      A     M      0.2;
      =     L     22.0;
      BLD   103;
      AN    M      3.3;
      =     L     22.1;
      BLD   103;
      CALL FB    12 , DB    72 (
           REQ                      := L     22.0,
           R                        := L     22.1,
           ID                       := W#16#12,
           R_ID                     := DW#16#12,
           DONE                     := DB2.DBX   10.0,
           ERROR                    := DB2.DBX   10.1,
           STATUS                   := DB2.DBW   12,
           SD_1                     := DB16.SHUTTLE,
           LEN                      := #SEND2_LEN);
      NOP   0;
NETWORK
TITLE =

      L     20;
      T     #RECV3_LEN;
      NOP   0;
NETWORK
TITLE =LOCAL(CPU4) --> LOCAL(CPU3) 공정상태
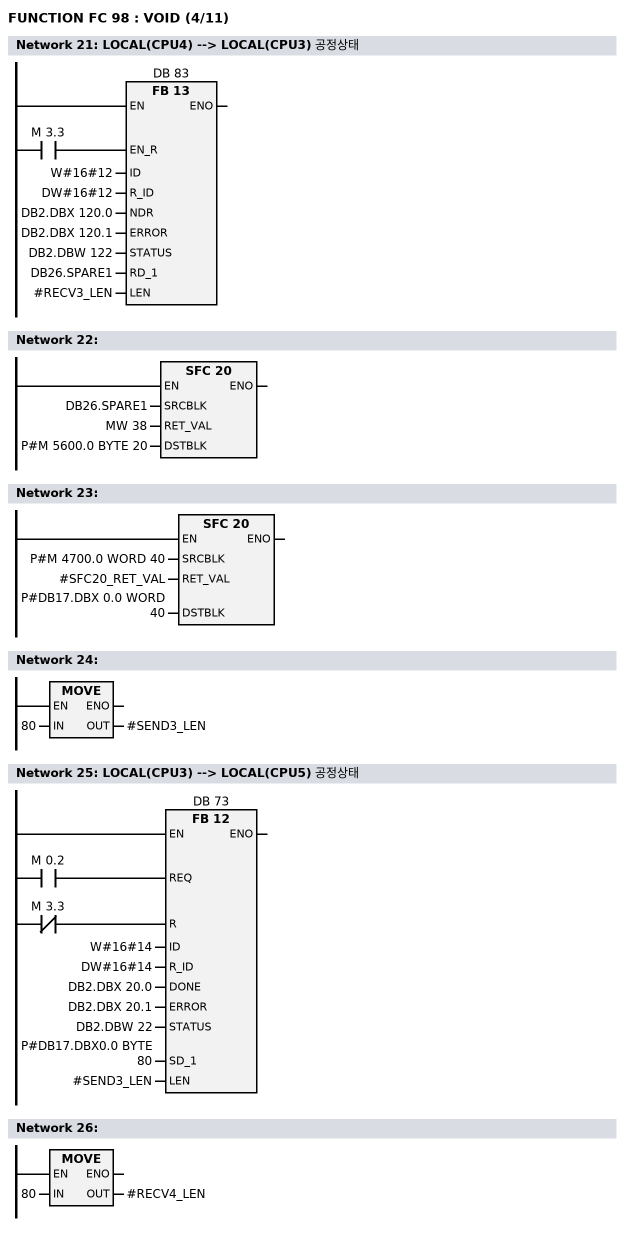

      A     M      3.3;
      =     L     22.0;
      BLD   103;
      CALL FB    13 , DB    83 (
           EN_R                     := L     22.0,
           ID                       := W#16#12,
           R_ID                     := DW#16#12,
           NDR                      := DB2.DBX  120.0,
           ERROR                    := DB2.DBX  120.1,
           STATUS                   := DB2.DBW  122,
           RD_1                     := DB26.SPARE1,
           LEN                      := #RECV3_LEN);
      NOP   0;
NETWORK
TITLE =

      CALL SFC   20 (
           SRCBLK                   := DB26.SPARE1,
           RET_VAL                  := MW    38,
           DSTBLK                   := P#M 5600.0 BYTE 20);
      NOP   0;
NETWORK
TITLE =

      CALL SFC   20 (
           SRCBLK                   := P#M 4700.0 WORD 40,
           RET_VAL                  := #SFC20_RET_VAL,
           DSTBLK                   := P#DB17.DBX 0.0 WORD 40);
      NOP   0;
NETWORK
TITLE =

      L     80;
      T     #SEND3_LEN;
      NOP   0;
NETWORK
TITLE =LOCAL(CPU3) --> LOCAL(CPU5) 공정상태

      A     M      0.2;
      =     L     22.0;
      BLD   103;
      AN    M      3.3;
      =     L     22.1;
      BLD   103;
      CALL FB    12 , DB    73 (
           REQ                      := L     22.0,
           R                        := L     22.1,
           ID                       := W#16#14,
           R_ID                     := DW#16#14,
           DONE                     := DB2.DBX   20.0,
           ERROR                    := DB2.DBX   20.1,
           STATUS                   := DB2.DBW   22,
           SD_1                     := P#DB17.DBX0.0 BYTE 80,
           LEN                      := #SEND3_LEN);
      NOP   0;
NETWORK
TITLE =

      L     80;
      T     #RECV4_LEN;
      NOP   0;
NETWORK
TITLE =LOCAL(CPU5) --> LOCAL(CPU3) 공정상태
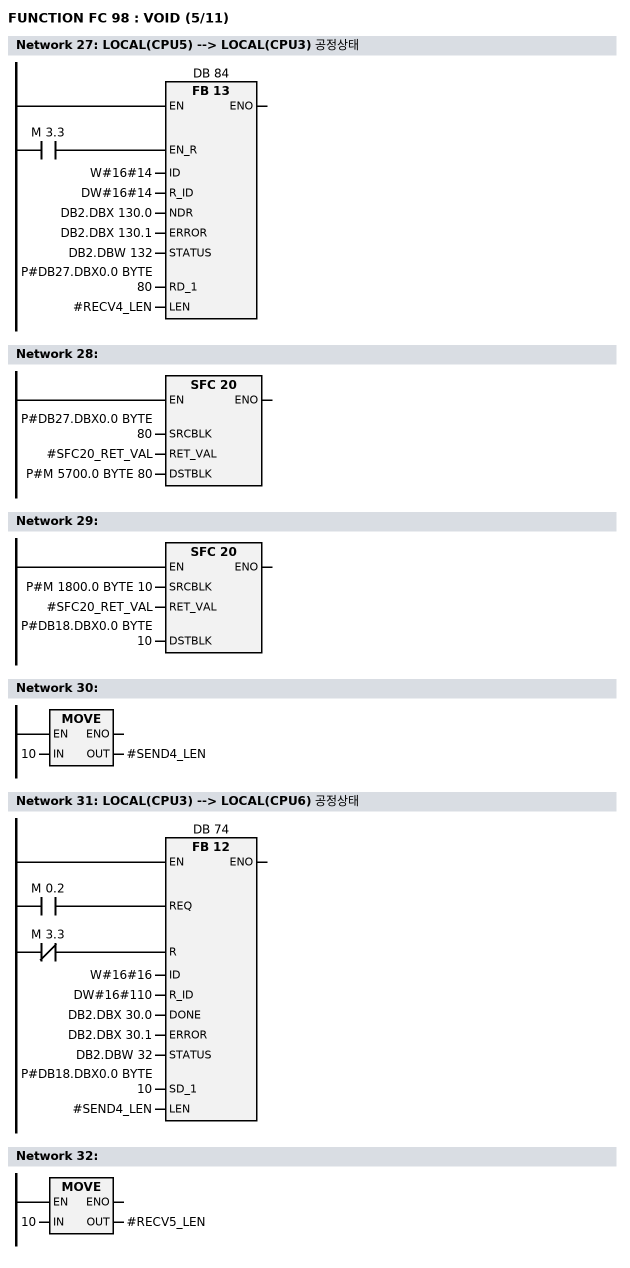

      A     M      3.3;
      =     L     22.0;
      BLD   103;
      CALL FB    13 , DB    84 (
           EN_R                     := L     22.0,
           ID                       := W#16#14,
           R_ID                     := DW#16#14,
           NDR                      := DB2.DBX  130.0,
           ERROR                    := DB2.DBX  130.1,
           STATUS                   := DB2.DBW  132,
           RD_1                     := P#DB27.DBX0.0 BYTE 80,
           LEN                      := #RECV4_LEN);
      NOP   0;
NETWORK
TITLE =

      CALL SFC   20 (
           SRCBLK                   := P#DB27.DBX0.0 BYTE 80,
           RET_VAL                  := #SFC20_RET_VAL,
           DSTBLK                   := P#M 5700.0 BYTE 80);
      NOP   0;
NETWORK
TITLE =

      CALL SFC   20 (
           SRCBLK                   := P#M 1800.0 BYTE 10,
           RET_VAL                  := #SFC20_RET_VAL,
           DSTBLK                   := P#DB18.DBX0.0 BYTE 10);
      NOP   0;
NETWORK
TITLE =

      L     10;
      T     #SEND4_LEN;
      NOP   0;
NETWORK
TITLE =LOCAL(CPU3) --> LOCAL(CPU6) 공정상태

      A     M      0.2;
      =     L     22.0;
      BLD   103;
      AN    M      3.3;
      =     L     22.1;
      BLD   103;
      CALL FB    12 , DB    74 (
           REQ                      := L     22.0,
           R                        := L     22.1,
           ID                       := W#16#16,
           R_ID                     := DW#16#110,
           DONE                     := DB2.DBX   30.0,
           ERROR                    := DB2.DBX   30.1,
           STATUS                   := DB2.DBW   32,
           SD_1                     := P#DB18.DBX0.0 BYTE 10,
           LEN                      := #SEND4_LEN);
      NOP   0;
NETWORK
TITLE =

      L     10;
      T     #RECV5_LEN;
      NOP   0;
NETWORK
TITLE =LOCAL(CPU6) --> LOCAL(CPU3) 공정상태
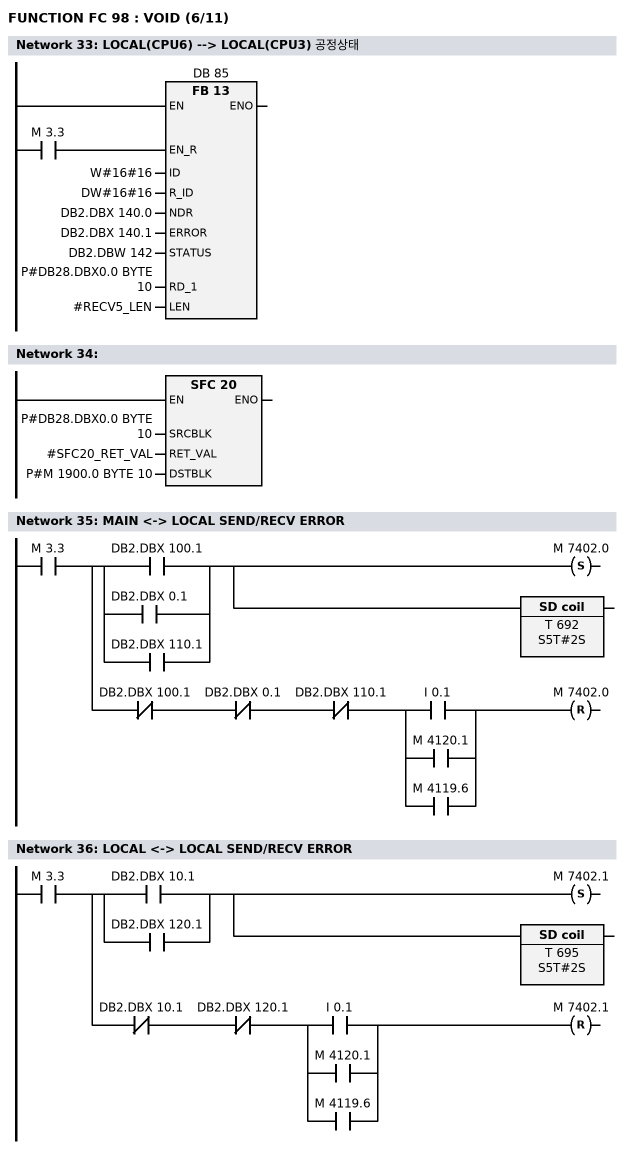

      A     M      3.3;
      =     L     22.0;
      BLD   103;
      CALL FB    13 , DB    85 (
           EN_R                     := L     22.0,
           ID                       := W#16#16,
           R_ID                     := DW#16#16,
           NDR                      := DB2.DBX  140.0,
           ERROR                    := DB2.DBX  140.1,
           STATUS                   := DB2.DBW  142,
           RD_1                     := P#DB28.DBX0.0 BYTE 10,
           LEN                      := #RECV5_LEN);
      NOP   0;
NETWORK
TITLE =

      CALL SFC   20 (
           SRCBLK                   := P#DB28.DBX0.0 BYTE 10,
           RET_VAL                  := #SFC20_RET_VAL,
           DSTBLK                   := P#M 1900.0 BYTE 10);
      NOP   0;
NETWORK
TITLE =MAIN <-> LOCAL SEND/RECV ERROR

      A     M      3.3;
      =     L     22.0;
      A     L     22.0;
      A(    ;
      O     DB2.DBX  100.1;
      O     DB2.DBX    0.1;
      O     DB2.DBX  110.1;
      )     ;
      S     M   7402.0;
      L     S5T#2S;
      SD    T    692;
      A     L     22.0;
      AN    DB2.DBX  100.1;
      AN    DB2.DBX    0.1;
      AN    DB2.DBX  110.1;
      A(    ;
      O     I      0.1;
      O     M   4120.1;
      O     M   4119.6;
      )     ;
      R     M   7402.0;
NETWORK
TITLE =LOCAL <-> LOCAL SEND/RECV ERROR

      A     M      3.3;
      =     L     22.0;
      A     L     22.0;
      A(    ;
      O     DB2.DBX   10.1;
      O     DB2.DBX  120.1;
      )     ;
      S     M   7402.1;
      L     S5T#2S;
      SD    T    695;
      A     L     22.0;
      AN    DB2.DBX   10.1;
      AN    DB2.DBX  120.1;
      A(    ;
      O     I      0.1;
      O     M   4120.1;
      O     M   4119.6;
      )     ;
      R     M   7402.1;
NETWORK
TITLE =LOCAL <-> LOCAL SEND/RECV ERROR
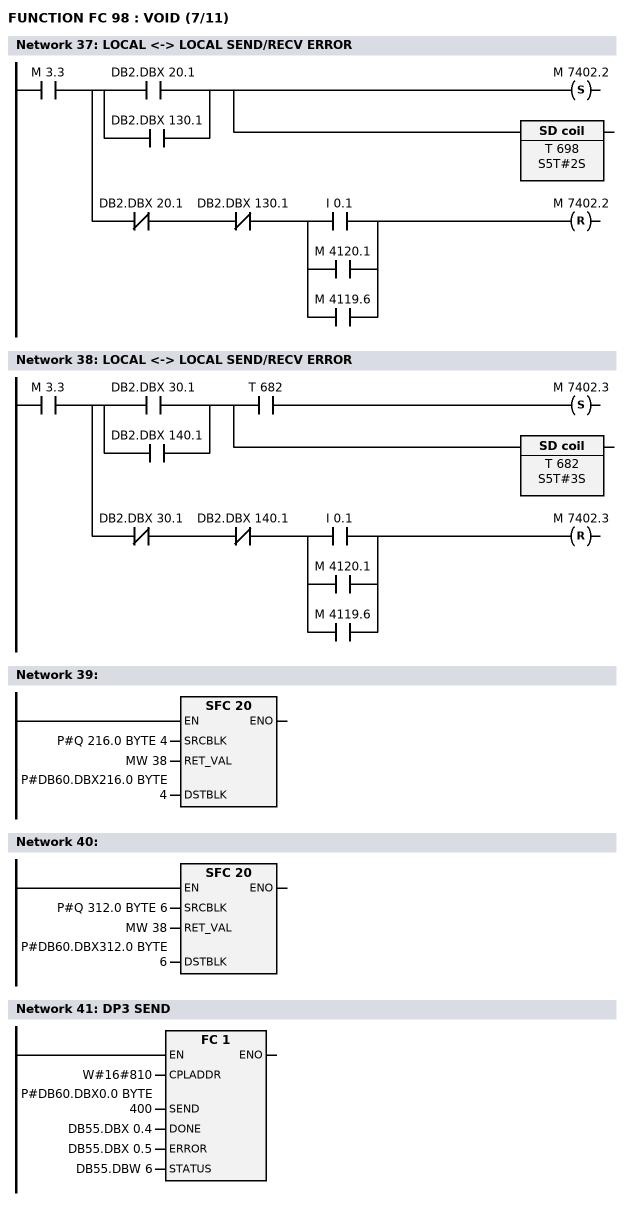

      A     M      3.3;
      =     L     22.0;
      A     L     22.0;
      A(    ;
      O     DB2.DBX   20.1;
      O     DB2.DBX  130.1;
      )     ;
      S     M   7402.2;
      L     S5T#2S;
      SD    T    698;
      A     L     22.0;
      AN    DB2.DBX   20.1;
      AN    DB2.DBX  130.1;
      A(    ;
      O     I      0.1;
      O     M   4120.1;
      O     M   4119.6;
      )     ;
      R     M   7402.2;
NETWORK
TITLE =LOCAL <-> LOCAL SEND/RECV ERROR

      A     M      3.3;
      =     L     22.0;
      A     L     22.0;
      A(    ;
      O     DB2.DBX   30.1;
      O     DB2.DBX  140.1;
      )     ;
      =     L     22.1;
      A     L     22.1;
      A     T    682;
      S     M   7402.3;
      A     L     22.1;
      BLD   102;
      L     S5T#3S;
      SD    T    682;
      A     L     22.0;
      AN    DB2.DBX   30.1;
      AN    DB2.DBX  140.1;
      A(    ;
      O     I      0.1;
      O     M   4120.1;
      O     M   4119.6;
      )     ;
      R     M   7402.3;
NETWORK
TITLE =

      CALL SFC   20 (
           SRCBLK                   := P#Q 216.0 BYTE 4,
           RET_VAL                  := MW    38,
           DSTBLK                   := P#DB60.DBX216.0 BYTE 4);
      NOP   0;
NETWORK
TITLE =

      CALL SFC   20 (
           SRCBLK                   := P#Q 312.0 BYTE 6,
           RET_VAL                  := MW    38,
           DSTBLK                   := P#DB60.DBX312.0 BYTE 6);
      NOP   0;
NETWORK
TITLE =DP3 SEND

      CALL FC     1 (
           CPLADDR                  := W#16#810,
           SEND                     := P#DB60.DBX0.0 BYTE 400,
           DONE                     := DB55.DBX    0.4,
           ERROR                    := DB55.DBX    0.5,
           STATUS                   := DB55.DBW    6);
      NOP   0;
NETWORK
TITLE =DP3 RECV
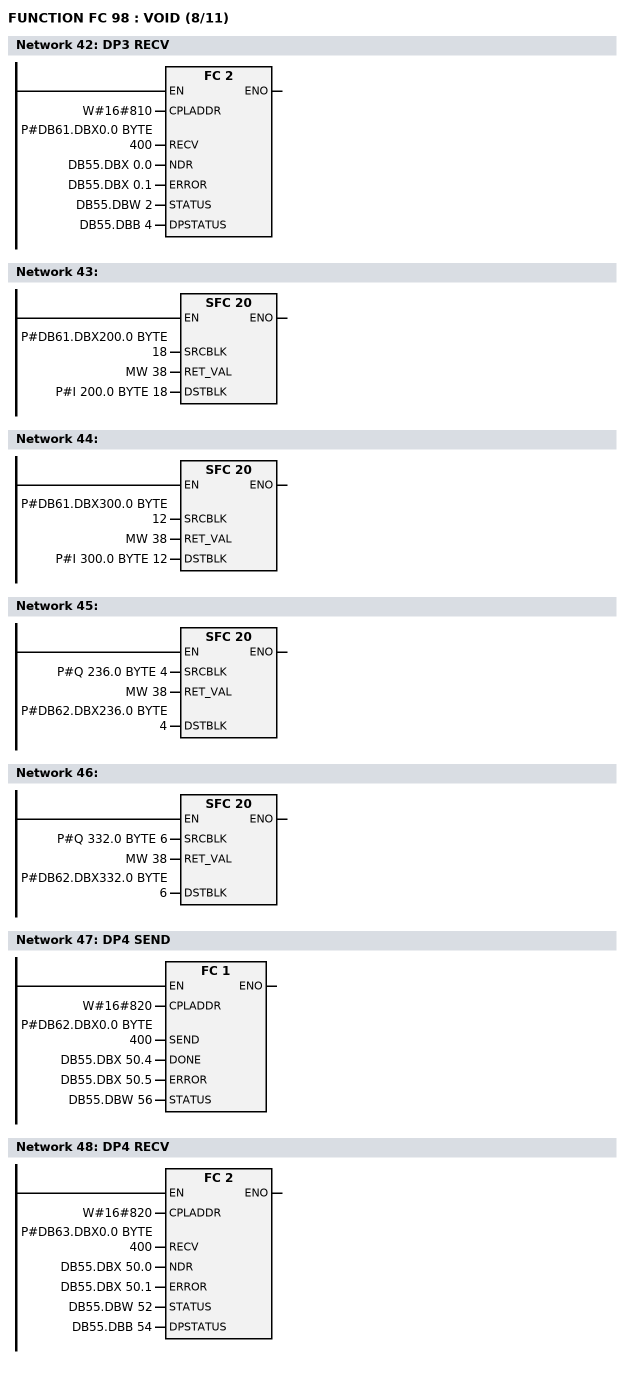

      CALL FC     2 (
           CPLADDR                  := W#16#810,
           RECV                     := P#DB61.DBX0.0 BYTE 400,
           NDR                      := DB55.DBX    0.0,
           ERROR                    := DB55.DBX    0.1,
           STATUS                   := DB55.DBW    2,
           DPSTATUS                 := DB55.DBB    4);
      NOP   0;
NETWORK
TITLE =

      CALL SFC   20 (
           SRCBLK                   := P#DB61.DBX200.0 BYTE 18,
           RET_VAL                  := MW    38,
           DSTBLK                   := P#I 200.0 BYTE 18);
      NOP   0;
NETWORK
TITLE =

      CALL SFC   20 (
           SRCBLK                   := P#DB61.DBX300.0 BYTE 12,
           RET_VAL                  := MW    38,
           DSTBLK                   := P#I 300.0 BYTE 12);
      NOP   0;
NETWORK
TITLE =

      CALL SFC   20 (
           SRCBLK                   := P#Q 236.0 BYTE 4,
           RET_VAL                  := MW    38,
           DSTBLK                   := P#DB62.DBX236.0 BYTE 4);
      NOP   0;
NETWORK
TITLE =

      CALL SFC   20 (
           SRCBLK                   := P#Q 332.0 BYTE 6,
           RET_VAL                  := MW    38,
           DSTBLK                   := P#DB62.DBX332.0 BYTE 6);
      NOP   0;
NETWORK
TITLE =DP4 SEND

      CALL FC     1 (
           CPLADDR                  := W#16#820,
           SEND                     := P#DB62.DBX0.0 BYTE 400,
           DONE                     := DB55.DBX   50.4,
           ERROR                    := DB55.DBX   50.5,
           STATUS                   := DB55.DBW   56);
      NOP   0;
NETWORK
TITLE =DP4 RECV

      CALL FC     2 (
           CPLADDR                  := W#16#820,
           RECV                     := P#DB63.DBX0.0 BYTE 400,
           NDR                      := DB55.DBX   50.0,
           ERROR                    := DB55.DBX   50.1,
           STATUS                   := DB55.DBW   52,
           DPSTATUS                 := DB55.DBB   54);
      NOP   0;
NETWORK
TITLE =
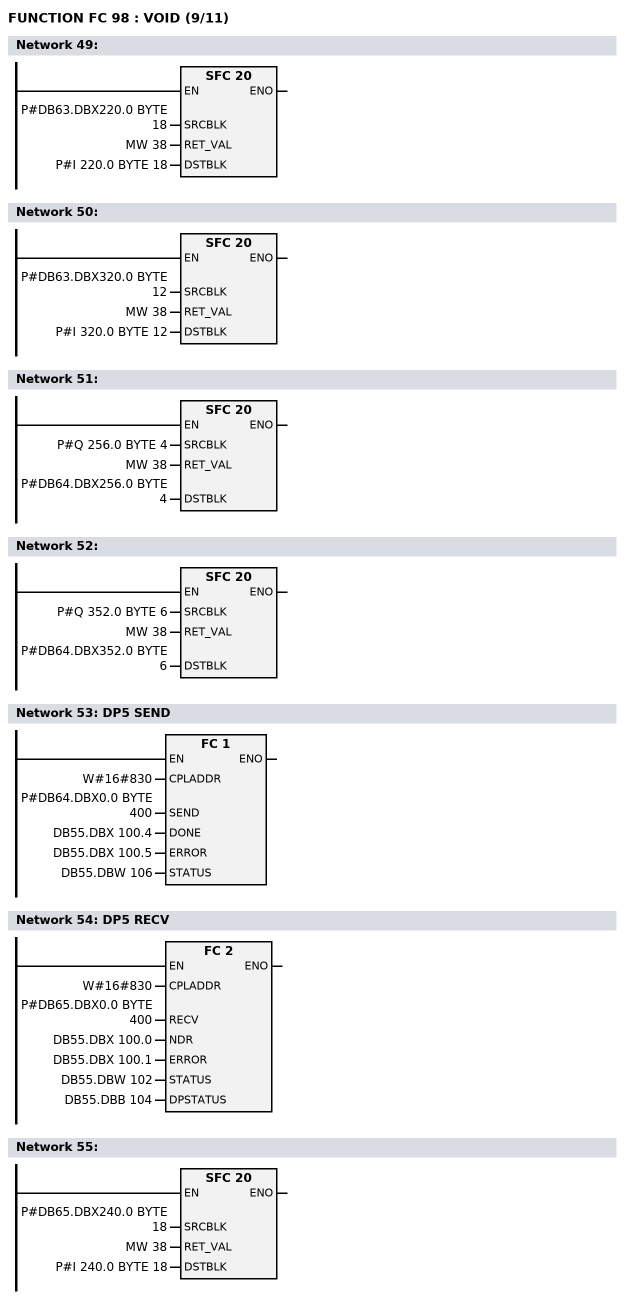

      CALL SFC   20 (
           SRCBLK                   := P#DB63.DBX220.0 BYTE 18,
           RET_VAL                  := MW    38,
           DSTBLK                   := P#I 220.0 BYTE 18);
      NOP   0;
NETWORK
TITLE =

      CALL SFC   20 (
           SRCBLK                   := P#DB63.DBX320.0 BYTE 12,
           RET_VAL                  := MW    38,
           DSTBLK                   := P#I 320.0 BYTE 12);
      NOP   0;
NETWORK
TITLE =

      CALL SFC   20 (
           SRCBLK                   := P#Q 256.0 BYTE 4,
           RET_VAL                  := MW    38,
           DSTBLK                   := P#DB64.DBX256.0 BYTE 4);
      NOP   0;
NETWORK
TITLE =

      CALL SFC   20 (
           SRCBLK                   := P#Q 352.0 BYTE 6,
           RET_VAL                  := MW    38,
           DSTBLK                   := P#DB64.DBX352.0 BYTE 6);
      NOP   0;
NETWORK
TITLE =DP5 SEND

      CALL FC     1 (
           CPLADDR                  := W#16#830,
           SEND                     := P#DB64.DBX0.0 BYTE 400,
           DONE                     := DB55.DBX  100.4,
           ERROR                    := DB55.DBX  100.5,
           STATUS                   := DB55.DBW  106);
      NOP   0;
NETWORK
TITLE =DP5 RECV

      CALL FC     2 (
           CPLADDR                  := W#16#830,
           RECV                     := P#DB65.DBX0.0 BYTE 400,
           NDR                      := DB55.DBX  100.0,
           ERROR                    := DB55.DBX  100.1,
           STATUS                   := DB55.DBW  102,
           DPSTATUS                 := DB55.DBB  104);
      NOP   0;
NETWORK
TITLE =

      CALL SFC   20 (
           SRCBLK                   := P#DB65.DBX240.0 BYTE 18,
           RET_VAL                  := MW    38,
           DSTBLK                   := P#I 240.0 BYTE 18);
      NOP   0;
NETWORK
TITLE =
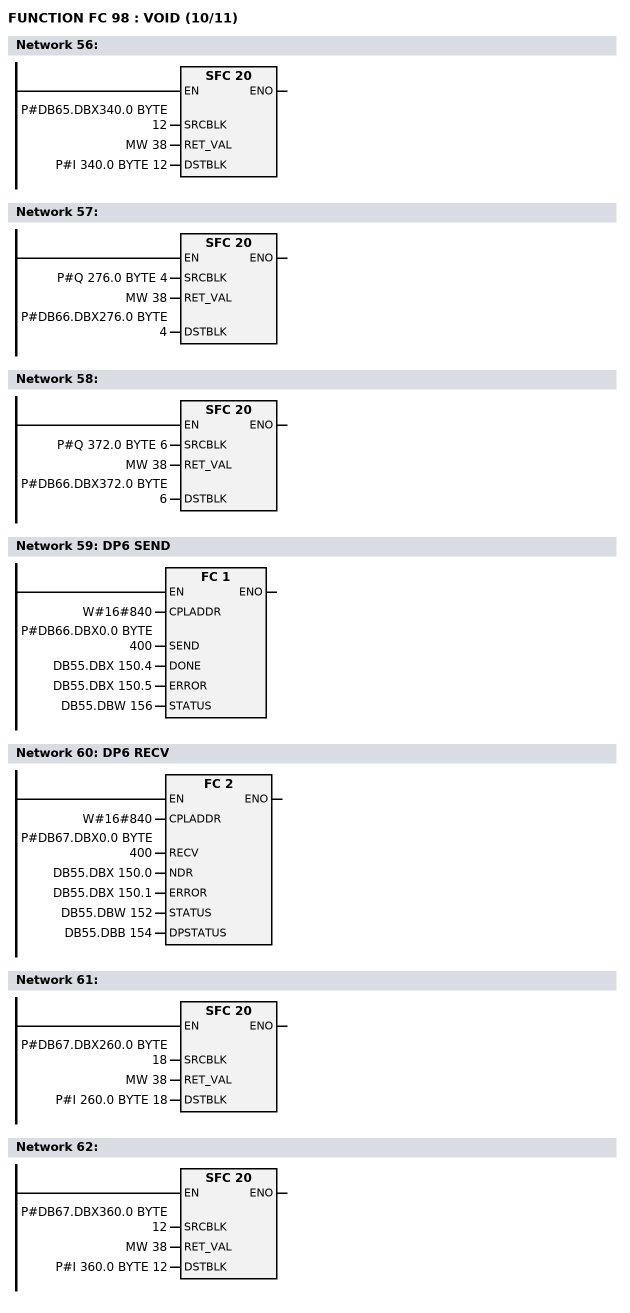

      CALL SFC   20 (
           SRCBLK                   := P#DB65.DBX340.0 BYTE 12,
           RET_VAL                  := MW    38,
           DSTBLK                   := P#I 340.0 BYTE 12);
      NOP   0;
NETWORK
TITLE =

      CALL SFC   20 (
           SRCBLK                   := P#Q 276.0 BYTE 4,
           RET_VAL                  := MW    38,
           DSTBLK                   := P#DB66.DBX276.0 BYTE 4);
      NOP   0;
NETWORK
TITLE =

      CALL SFC   20 (
           SRCBLK                   := P#Q 372.0 BYTE 6,
           RET_VAL                  := MW    38,
           DSTBLK                   := P#DB66.DBX372.0 BYTE 6);
      NOP   0;
NETWORK
TITLE =DP6 SEND

      CALL FC     1 (
           CPLADDR                  := W#16#840,
           SEND                     := P#DB66.DBX0.0 BYTE 400,
           DONE                     := DB55.DBX  150.4,
           ERROR                    := DB55.DBX  150.5,
           STATUS                   := DB55.DBW  156);
      NOP   0;
NETWORK
TITLE =DP6 RECV

      CALL FC     2 (
           CPLADDR                  := W#16#840,
           RECV                     := P#DB67.DBX0.0 BYTE 400,
           NDR                      := DB55.DBX  150.0,
           ERROR                    := DB55.DBX  150.1,
           STATUS                   := DB55.DBW  152,
           DPSTATUS                 := DB55.DBB  154);
      NOP   0;
NETWORK
TITLE =

      CALL SFC   20 (
           SRCBLK                   := P#DB67.DBX260.0 BYTE 18,
           RET_VAL                  := MW    38,
           DSTBLK                   := P#I 260.0 BYTE 18);
      NOP   0;
NETWORK
TITLE =

      CALL SFC   20 (
           SRCBLK                   := P#DB67.DBX360.0 BYTE 12,
           RET_VAL                  := MW    38,
           DSTBLK                   := P#I 360.0 BYTE 12);
      NOP   0;
NETWORK
TITLE =
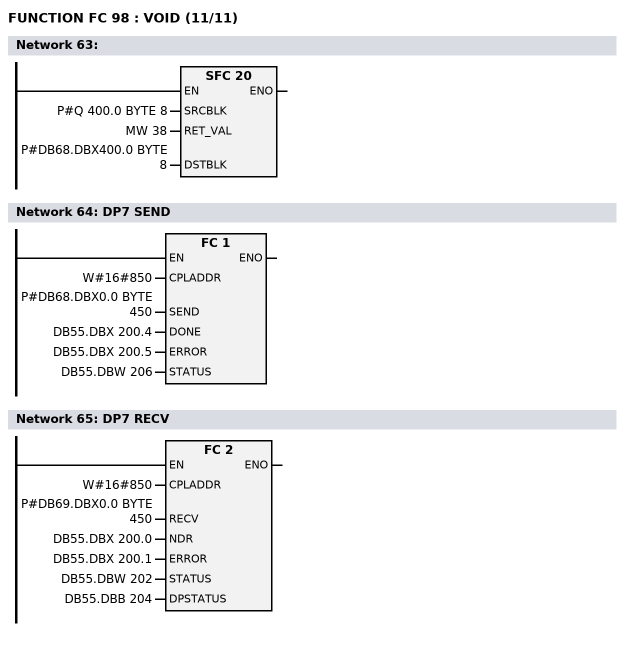

      CALL SFC   20 (
           SRCBLK                   := P#Q 400.0 BYTE 8,
           RET_VAL                  := MW    38,
           DSTBLK                   := P#DB68.DBX400.0 BYTE 8);
      NOP   0;
NETWORK
TITLE =DP7 SEND

      CALL FC     1 (
           CPLADDR                  := W#16#850,
           SEND                     := P#DB68.DBX0.0 BYTE 450,
           DONE                     := DB55.DBX  200.4,
           ERROR                    := DB55.DBX  200.5,
           STATUS                   := DB55.DBW  206);
      NOP   0;
NETWORK
TITLE =DP7 RECV

      CALL FC     2 (
           CPLADDR                  := W#16#850,
           RECV                     := P#DB69.DBX0.0 BYTE 450,
           NDR                      := DB55.DBX  200.0,
           ERROR                    := DB55.DBX  200.1,
           STATUS                   := DB55.DBW  202,
           DPSTATUS                 := DB55.DBB  204);
      NOP   0;
END_FUNCTION

FUNCTION FC 100 : VOID
TITLE =
VERSION : 0.1

BEGIN
NETWORK
TITLE =
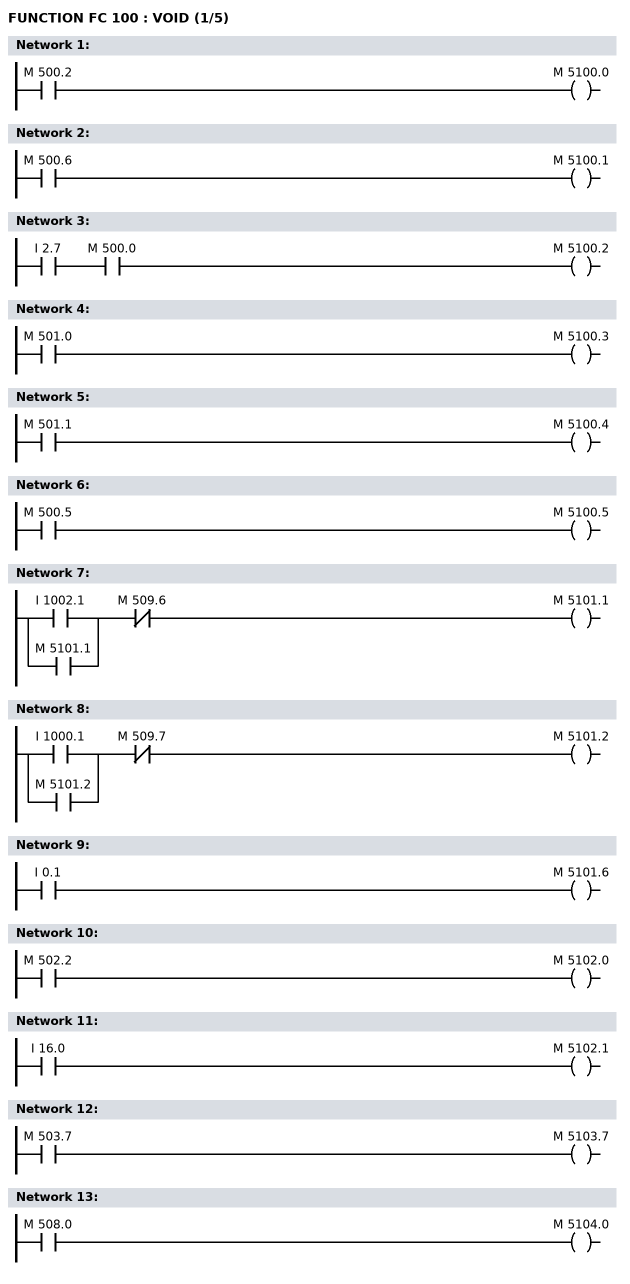

      A     M    500.2;
      =     M   5100.0;
NETWORK
TITLE =

      A     M    500.6;
      =     M   5100.1;
NETWORK
TITLE =

      A     I      2.7;
      A     M    500.0;
      =     M   5100.2;
NETWORK
TITLE =

      A     M    501.0;
      =     M   5100.3;
NETWORK
TITLE =

      A     M    501.1;
      =     M   5100.4;
NETWORK
TITLE =

      A     M    500.5;
      =     M   5100.5;
NETWORK
TITLE =

      A(    ;
      O     I   1002.1;
      O     M   5101.1;
      )     ;
      AN    M    509.6;
      =     M   5101.1;
NETWORK
TITLE =

      A(    ;
      O     I   1000.1;
      O     M   5101.2;
      )     ;
      AN    M    509.7;
      =     M   5101.2;
NETWORK
TITLE =

      A     I      0.1;
      =     M   5101.6;
NETWORK
TITLE =

      A     M    502.2;
      =     M   5102.0;
NETWORK
TITLE =

      A     I     16.0;
      =     M   5102.1;
NETWORK
TITLE =

      A     M    503.7;
      =     M   5103.7;
NETWORK
TITLE =

      A     M    508.0;
      =     M   5104.0;
NETWORK
TITLE =
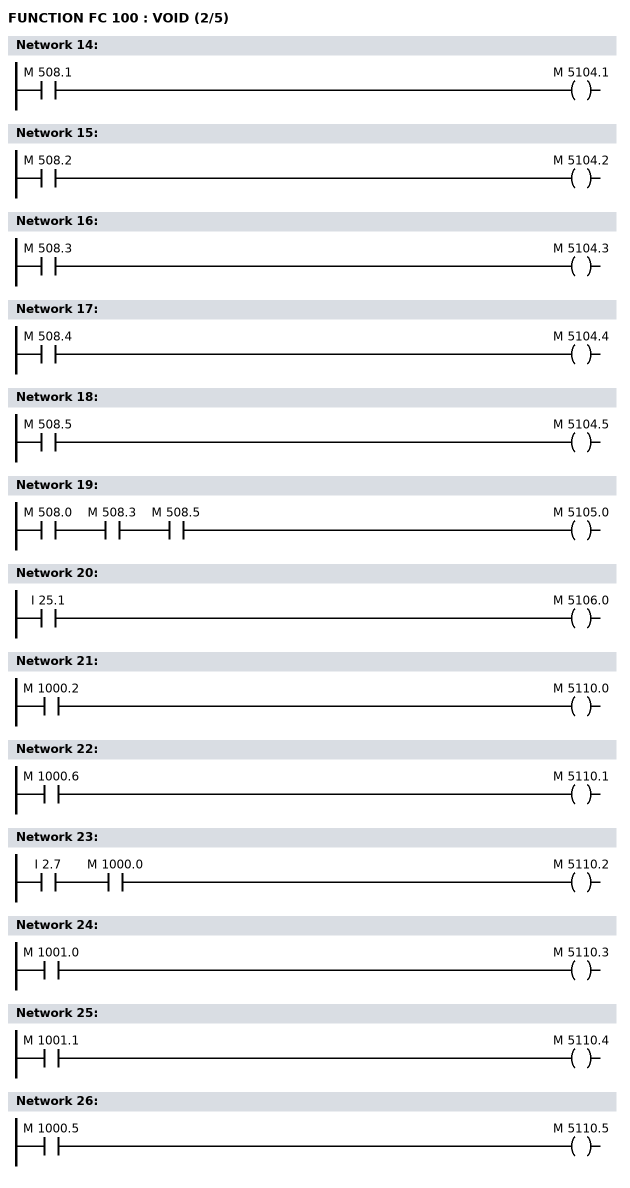

      A     M    508.1;
      =     M   5104.1;
NETWORK
TITLE =

      A     M    508.2;
      =     M   5104.2;
NETWORK
TITLE =

      A     M    508.3;
      =     M   5104.3;
NETWORK
TITLE =

      A     M    508.4;
      =     M   5104.4;
NETWORK
TITLE =

      A     M    508.5;
      =     M   5104.5;
NETWORK
TITLE =

      A     M    508.0;
      A     M    508.3;
      A     M    508.5;
      =     M   5105.0;
NETWORK
TITLE =

      A     I     25.1;
      =     M   5106.0;
NETWORK
TITLE =

      A     M   1000.2;
      =     M   5110.0;
NETWORK
TITLE =

      A     M   1000.6;
      =     M   5110.1;
NETWORK
TITLE =

      A     I      2.7;
      A     M   1000.0;
      =     M   5110.2;
NETWORK
TITLE =

      A     M   1001.0;
      =     M   5110.3;
NETWORK
TITLE =

      A     M   1001.1;
      =     M   5110.4;
NETWORK
TITLE =

      A     M   1000.5;
      =     M   5110.5;
NETWORK
TITLE =
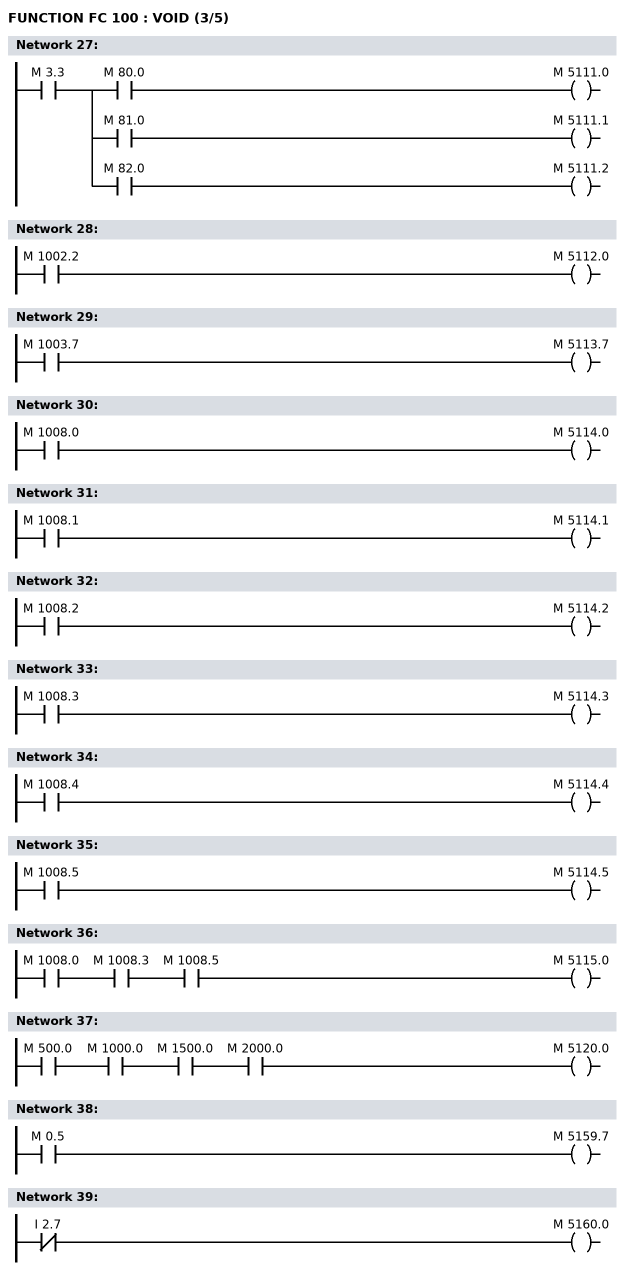

      A     M      3.3;
      =     L      0.0;
      A     L      0.0;
      A     M     80.0;
      =     M   5111.0;
      A     L      0.0;
      A     M     81.0;
      =     M   5111.1;
      A     L      0.0;
      A     M     82.0;
      =     M   5111.2;
NETWORK
TITLE =

      A     M   1002.2;
      =     M   5112.0;
NETWORK
TITLE =

      A     M   1003.7;
      =     M   5113.7;
NETWORK
TITLE =

      A     M   1008.0;
      =     M   5114.0;
NETWORK
TITLE =

      A     M   1008.1;
      =     M   5114.1;
NETWORK
TITLE =

      A     M   1008.2;
      =     M   5114.2;
NETWORK
TITLE =

      A     M   1008.3;
      =     M   5114.3;
NETWORK
TITLE =

      A     M   1008.4;
      =     M   5114.4;
NETWORK
TITLE =

      A     M   1008.5;
      =     M   5114.5;
NETWORK
TITLE =

      A     M   1008.0;
      A     M   1008.3;
      A     M   1008.5;
      =     M   5115.0;
NETWORK
TITLE =

      A     M    500.0;
      A     M   1000.0;
      A     M   1500.0;
      A     M   2000.0;
      =     M   5120.0;
NETWORK
TITLE =

      A     M      0.5;
      =     M   5159.7;
NETWORK
TITLE =

      AN    I      2.7;
      =     M   5160.0;
NETWORK
TITLE =
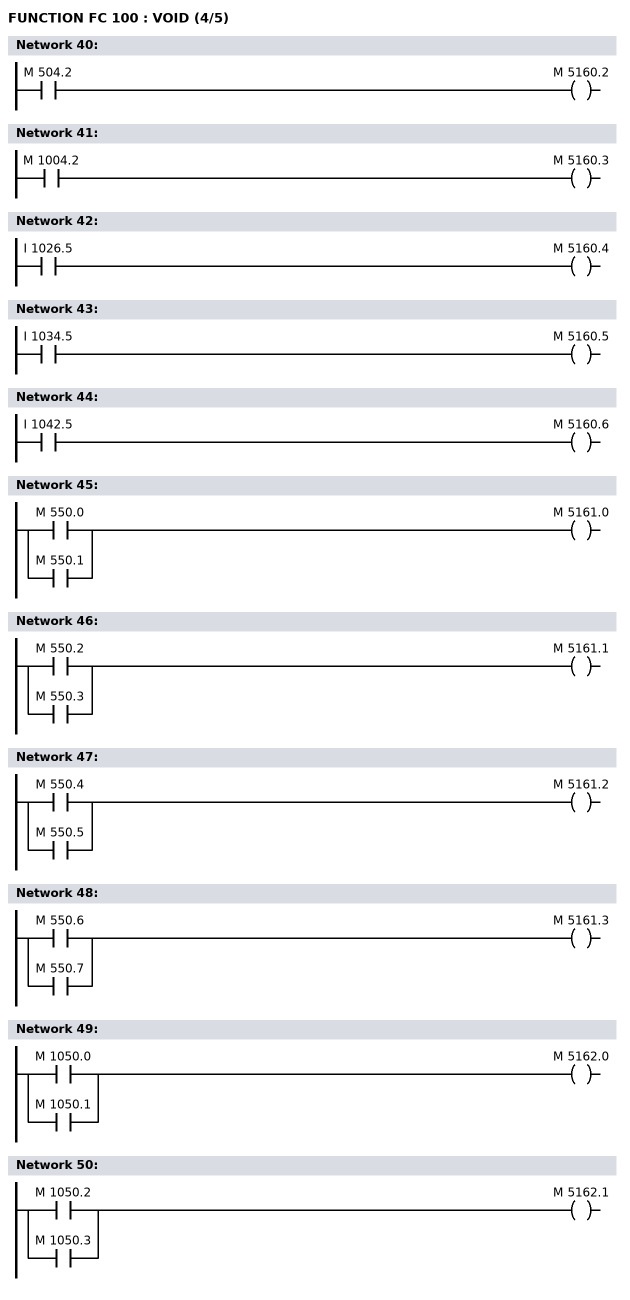

      A     M    504.2;
      =     M   5160.2;
NETWORK
TITLE =

      A     M   1004.2;
      =     M   5160.3;
NETWORK
TITLE =

      A     I   1026.5;
      =     M   5160.4;
NETWORK
TITLE =

      A     I   1034.5;
      =     M   5160.5;
NETWORK
TITLE =

      A     I   1042.5;
      =     M   5160.6;
NETWORK
TITLE =

      O     M    550.0;
      O     M    550.1;
      =     M   5161.0;
NETWORK
TITLE =

      O     M    550.2;
      O     M    550.3;
      =     M   5161.1;
NETWORK
TITLE =

      O     M    550.4;
      O     M    550.5;
      =     M   5161.2;
NETWORK
TITLE =

      O     M    550.6;
      O     M    550.7;
      =     M   5161.3;
NETWORK
TITLE =

      O     M   1050.0;
      O     M   1050.1;
      =     M   5162.0;
NETWORK
TITLE =

      O     M   1050.2;
      O     M   1050.3;
      =     M   5162.1;
NETWORK
TITLE =
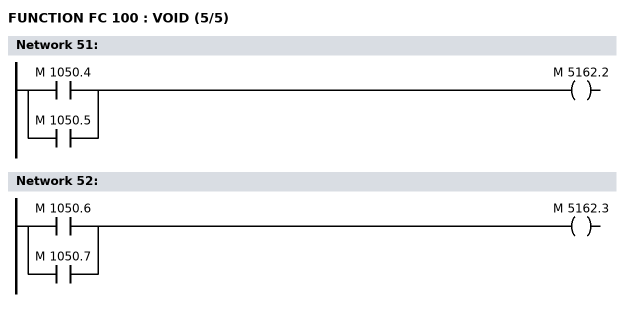

      O     M   1050.4;
      O     M   1050.5;
      =     M   5162.2;
NETWORK
TITLE =

      O     M   1050.6;
      O     M   1050.7;
      =     M   5162.3;
NETWORK
TITLE =

      AN    OV;
      =     L      0.0;
      A     L      0.0;
      A     M    503.0;
      =     M   5162.4;
      A     L      0.0;
      A     I      2.1;
      =     M   5162.5;
NETWORK
TITLE =
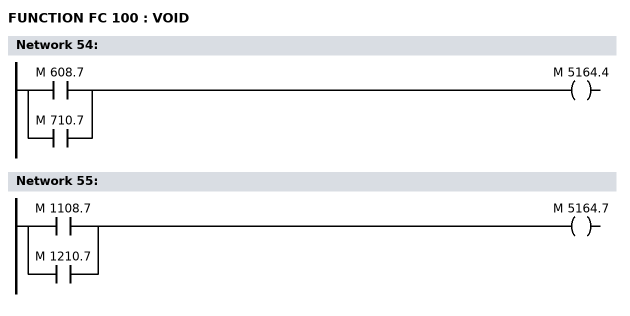

      O     M    608.7;
      O     M    710.7;
      =     M   5164.4;
NETWORK
TITLE =

      O     M   1108.7;
      O     M   1210.7;
      =     M   5164.7;
NETWORK
TITLE =

      AN    OV;
      =     L      0.0;
      A     L      0.0;
      AN    I   1003.0;
      =     M   5165.0;
      A     L      0.0;
      A     I   1003.1;
      =     M   5165.1;
      A     L      0.0;
      A     I   1003.2;
      =     M   5165.2;
      A     L      0.0;
      A     I   1003.4;
      =     M   5165.3;
      A     L      0.0;
      A     I   1003.5;
      =     M   5165.4;
      A     L      0.0;
      A     I   1003.6;
      =     M   5165.5;
      A     L      0.0;
      A     I   1003.7;
      =     M   5165.6;
      A     L      0.0;
      A     I   1002.7;
      =     M   5165.7;
NETWORK
TITLE =

      AN    OV;
      =     L      0.0;
      A     L      0.0;
      AN    I   1011.0;
      =     M   5166.0;
      A     L      0.0;
      A     I   1011.1;
      =     M   5166.1;
      A     L      0.0;
      A     I   1011.2;
      =     M   5166.2;
NETWORK
TITLE =

      AN    OV;
      =     L      0.0;
      A     L      0.0;
      A     M   1003.4;
      =     M   5166.3;
      A     L      0.0;
      A     M   1003.5;
      =     M   5166.4;
      A     L      0.0;
      A     M   1001.7;
      =     M   5166.5;
NETWORK
TITLE =
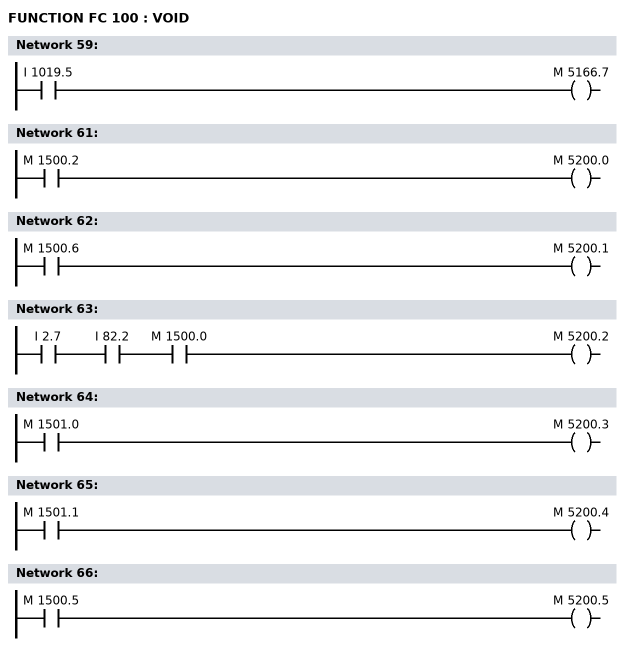

      A     I   1019.5;
      =     M   5166.7;
NETWORK
TITLE =

NETWORK
TITLE =

      A     M   1500.2;
      =     M   5200.0;
NETWORK
TITLE =

      A     M   1500.6;
      =     M   5200.1;
NETWORK
TITLE =

      A     I      2.7;
      A     I     82.2;
      A     M   1500.0;
      =     M   5200.2;
NETWORK
TITLE =

      A     M   1501.0;
      =     M   5200.3;
NETWORK
TITLE =

      A     M   1501.1;
      =     M   5200.4;
NETWORK
TITLE =

      A     M   1500.5;
      =     M   5200.5;
NETWORK
TITLE =

      A     M   2001.7;
      =     L      0.0;
      A     L      0.0;
      AN    M   2001.0;
      AN    M   2001.1;
      AN    M   2002.2;
      L     S5T#12S;
      SD    T    154;
      A     L      0.0;
      A     I     48.2;
      =     L      0.1;
      A     L      0.1;
      A     T    155;
      CU    C      1;
      A     L      0.1;
      BLD   102;
      L     S5T#8S;
      SD    T    155;
      A     L      0.0;
      A     I     48.3;
      =     L      0.1;
      A     L      0.1;
      A     T    156;
      CU    C      2;
      A     L      0.1;
      BLD   102;
      L     S5T#8S;
      SD    T    156;
      A     L      0.0;
      A     I     49.4;
      =     L      0.1;
      A     L      0.1;
      A     T    157;
      CU    C      3;
      A     L      0.1;
      BLD   102;
      L     S5T#8S;
      SD    T    157;
NETWORK
TITLE =
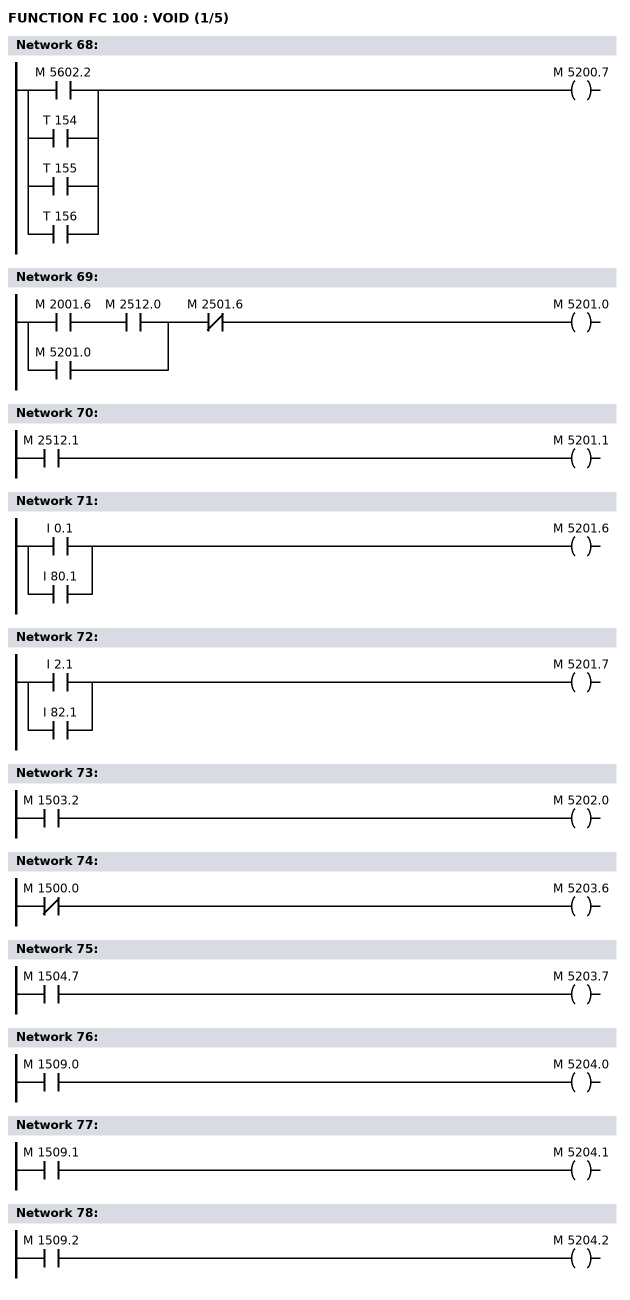

      O     M   5602.2;
      O     T    154;
      O     T    155;
      O     T    156;
      =     M   5200.7;
NETWORK
TITLE =

      A(    ;
      A     M   2001.6;
      A     M   2512.0;
      O     M   5201.0;
      )     ;
      AN    M   2501.6;
      =     M   5201.0;
NETWORK
TITLE =

      A     M   2512.1;
      =     M   5201.1;
NETWORK
TITLE =

      O     I      0.1;
      O     I     80.1;
      =     M   5201.6;
NETWORK
TITLE =

      O     I      2.1;
      O     I     82.1;
      =     M   5201.7;
NETWORK
TITLE =

      A     M   1503.2;
      =     M   5202.0;
NETWORK
TITLE =

      AN    M   1500.0;
      =     M   5203.6;
NETWORK
TITLE =

      A     M   1504.7;
      =     M   5203.7;
NETWORK
TITLE =

      A     M   1509.0;
      =     M   5204.0;
NETWORK
TITLE =

      A     M   1509.1;
      =     M   5204.1;
NETWORK
TITLE =

      A     M   1509.2;
      =     M   5204.2;
NETWORK
TITLE =
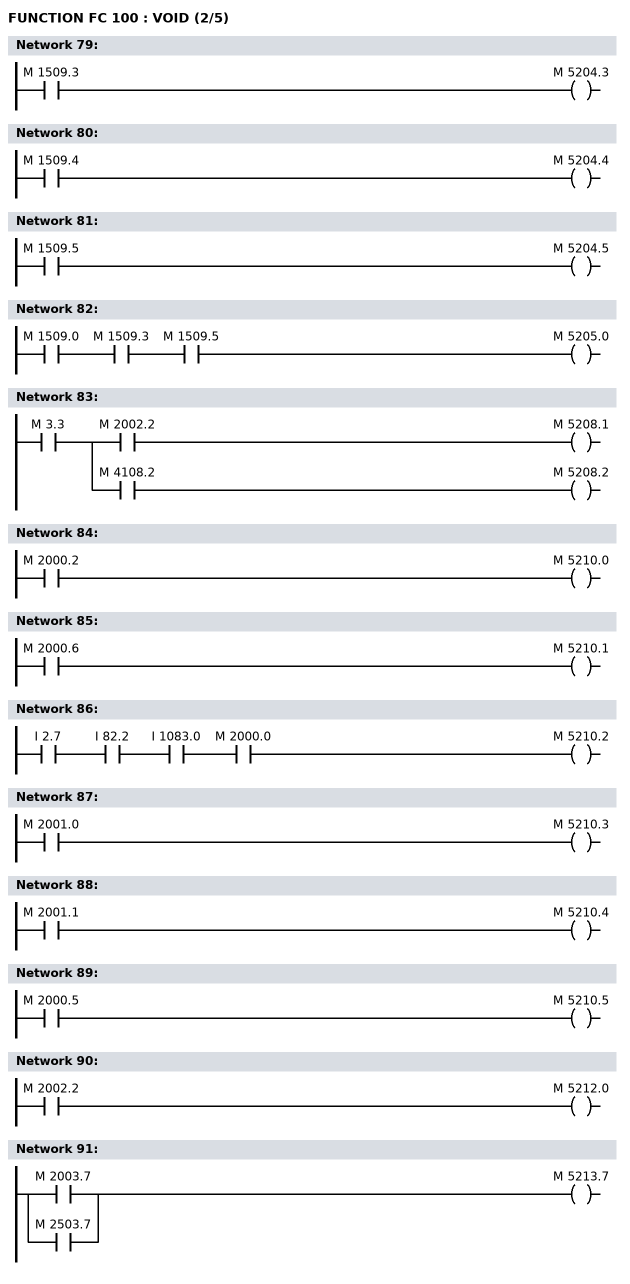

      A     M   1509.3;
      =     M   5204.3;
NETWORK
TITLE =

      A     M   1509.4;
      =     M   5204.4;
NETWORK
TITLE =

      A     M   1509.5;
      =     M   5204.5;
NETWORK
TITLE =

      A     M   1509.0;
      A     M   1509.3;
      A     M   1509.5;
      =     M   5205.0;
NETWORK
TITLE =

      A     M      3.3;
      =     L      0.0;
      A     L      0.0;
      A     M   2002.2;
      =     M   5208.1;
      A     L      0.0;
      A     M   4108.2;
      =     M   5208.2;
NETWORK
TITLE =

      A     M   2000.2;
      =     M   5210.0;
NETWORK
TITLE =

      A     M   2000.6;
      =     M   5210.1;
NETWORK
TITLE =

      A     I      2.7;
      A     I     82.2;
      A     I   1083.0;
      A     M   2000.0;
      =     M   5210.2;
NETWORK
TITLE =

      A     M   2001.0;
      =     M   5210.3;
NETWORK
TITLE =

      A     M   2001.1;
      =     M   5210.4;
NETWORK
TITLE =

      A     M   2000.5;
      =     M   5210.5;
NETWORK
TITLE =

      A     M   2002.2;
      =     M   5212.0;
NETWORK
TITLE =

      O     M   2003.7;
      O     M   2503.7;
      =     M   5213.7;
NETWORK
TITLE =
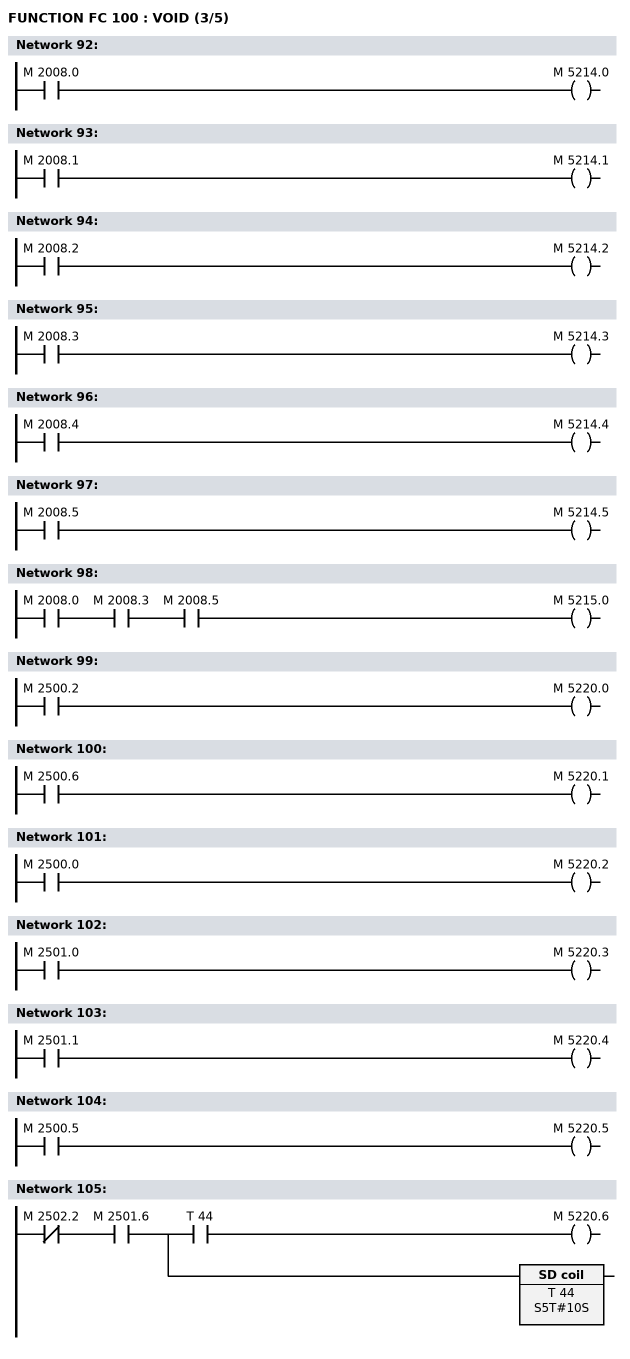

      A     M   2008.0;
      =     M   5214.0;
NETWORK
TITLE =

      A     M   2008.1;
      =     M   5214.1;
NETWORK
TITLE =

      A     M   2008.2;
      =     M   5214.2;
NETWORK
TITLE =

      A     M   2008.3;
      =     M   5214.3;
NETWORK
TITLE =

      A     M   2008.4;
      =     M   5214.4;
NETWORK
TITLE =

      A     M   2008.5;
      =     M   5214.5;
NETWORK
TITLE =

      A     M   2008.0;
      A     M   2008.3;
      A     M   2008.5;
      =     M   5215.0;
NETWORK
TITLE =

      A     M   2500.2;
      =     M   5220.0;
NETWORK
TITLE =

      A     M   2500.6;
      =     M   5220.1;
NETWORK
TITLE =

      A     M   2500.0;
      =     M   5220.2;
NETWORK
TITLE =

      A     M   2501.0;
      =     M   5220.3;
NETWORK
TITLE =

      A     M   2501.1;
      =     M   5220.4;
NETWORK
TITLE =

      A     M   2500.5;
      =     M   5220.5;
NETWORK
TITLE =

      AN    M   2502.2;
      A     M   2501.6;
      =     L      0.0;
      A     L      0.0;
      A     T     44;
      =     M   5220.6;
      A     L      0.0;
      BLD   102;
      L     S5T#10S;
      SD    T     44;
NETWORK
TITLE =
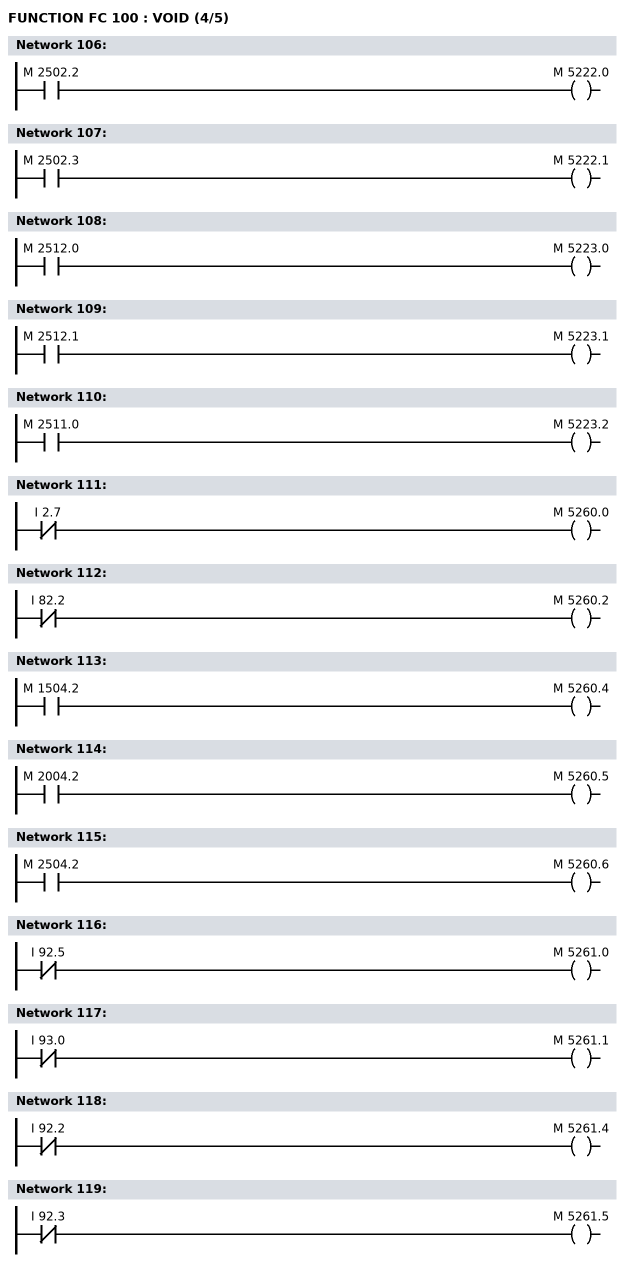

      A     M   2502.2;
      =     M   5222.0;
NETWORK
TITLE =

      A     M   2502.3;
      =     M   5222.1;
NETWORK
TITLE =

      A     M   2512.0;
      =     M   5223.0;
NETWORK
TITLE =

      A     M   2512.1;
      =     M   5223.1;
NETWORK
TITLE =

      A     M   2511.0;
      =     M   5223.2;
NETWORK
TITLE =

      AN    I      2.7;
      =     M   5260.0;
NETWORK
TITLE =

      AN    I     82.2;
      =     M   5260.2;
NETWORK
TITLE =

      A     M   1504.2;
      =     M   5260.4;
NETWORK
TITLE =

      A     M   2004.2;
      =     M   5260.5;
NETWORK
TITLE =

      A     M   2504.2;
      =     M   5260.6;
NETWORK
TITLE =

      AN    I     92.5;
      =     M   5261.0;
NETWORK
TITLE =

      AN    I     93.0;
      =     M   5261.1;
NETWORK
TITLE =

      AN    I     92.2;
      =     M   5261.4;
NETWORK
TITLE =

      AN    I     92.3;
      =     M   5261.5;
NETWORK
TITLE =
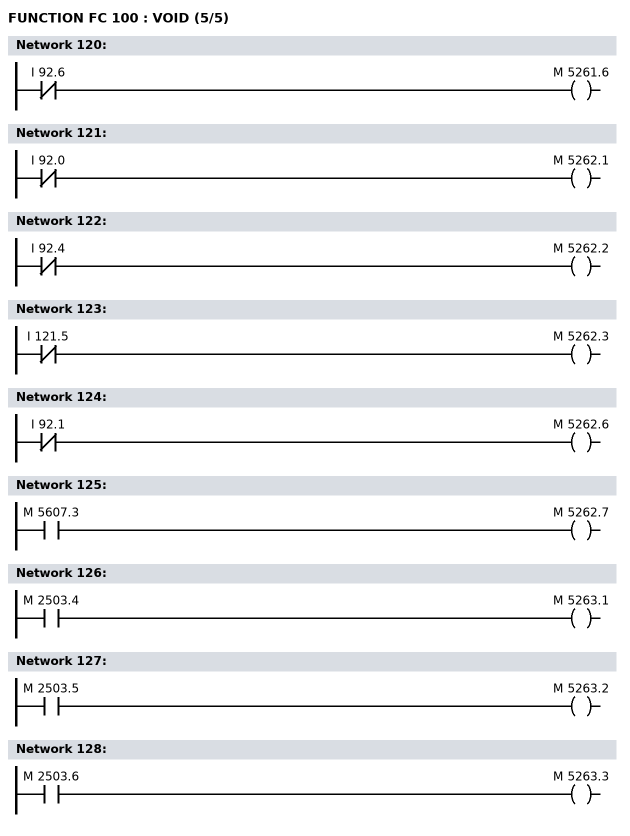

      AN    I     92.6;
      =     M   5261.6;
NETWORK
TITLE =

      AN    I     92.0;
      =     M   5262.1;
NETWORK
TITLE =

      AN    I     92.4;
      =     M   5262.2;
NETWORK
TITLE =

      AN    I    121.5;
      =     M   5262.3;
NETWORK
TITLE =

      AN    I     92.1;
      =     M   5262.6;
NETWORK
TITLE =

      A     M   5607.3;
      =     M   5262.7;
NETWORK
TITLE =

      A     M   2503.4;
      =     M   5263.1;
NETWORK
TITLE =

      A     M   2503.5;
      =     M   5263.2;
NETWORK
TITLE =

      A     M   2503.6;
      =     M   5263.3;
NETWORK
TITLE =

      AN    OV;
      AN    I     17.2;
      =     M   5263.4;
NETWORK
TITLE =
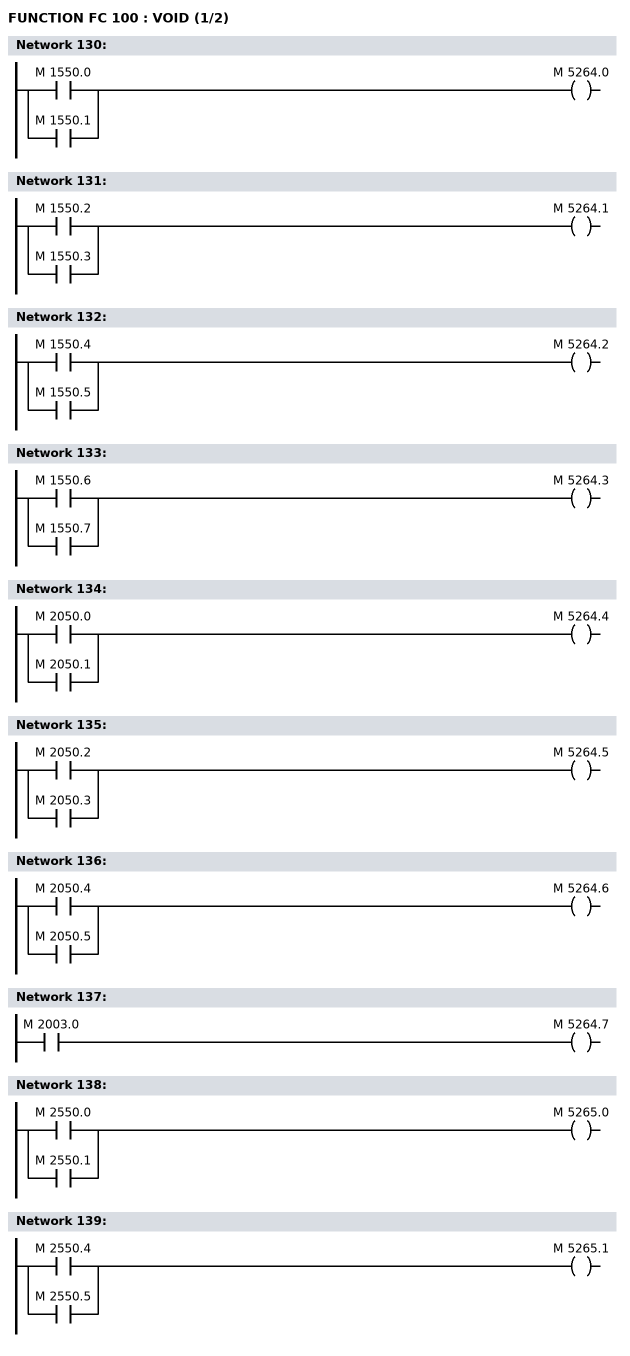

      O     M   1550.0;
      O     M   1550.1;
      =     M   5264.0;
NETWORK
TITLE =

      O     M   1550.2;
      O     M   1550.3;
      =     M   5264.1;
NETWORK
TITLE =

      O     M   1550.4;
      O     M   1550.5;
      =     M   5264.2;
NETWORK
TITLE =

      O     M   1550.6;
      O     M   1550.7;
      =     M   5264.3;
NETWORK
TITLE =

      O     M   2050.0;
      O     M   2050.1;
      =     M   5264.4;
NETWORK
TITLE =

      O     M   2050.2;
      O     M   2050.3;
      =     M   5264.5;
NETWORK
TITLE =

      O     M   2050.4;
      O     M   2050.5;
      =     M   5264.6;
NETWORK
TITLE =

      A     M   2003.0;
      =     M   5264.7;
NETWORK
TITLE =

      O     M   2550.0;
      O     M   2550.1;
      =     M   5265.0;
NETWORK
TITLE =

      O     M   2550.4;
      O     M   2550.5;
      =     M   5265.1;
NETWORK
TITLE =
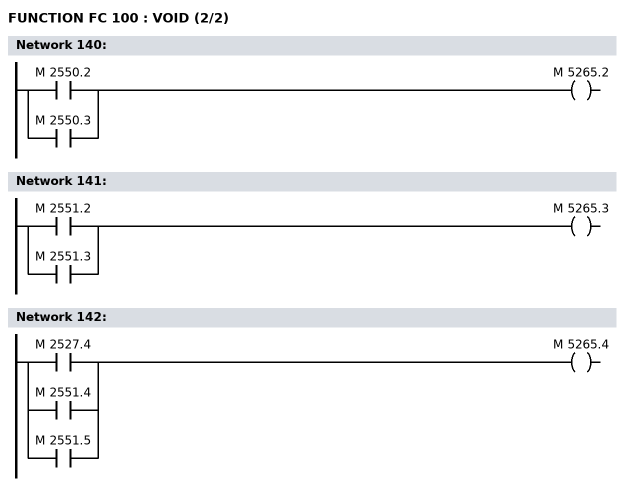

      O     M   2550.2;
      O     M   2550.3;
      =     M   5265.2;
NETWORK
TITLE =

      O     M   2551.2;
      O     M   2551.3;
      =     M   5265.3;
NETWORK
TITLE =

      O     M   2527.4;
      O     M   2551.4;
      O     M   2551.5;
      =     M   5265.4;
NETWORK
TITLE =

      AN    OV;
      =     L      0.0;
      A     L      0.0;
      A     I      2.1;
      =     M   5265.5;
      A     L      0.0;
      A     I     82.1;
      =     M   5265.6;
      A     L      0.0;
      A     M   2002.4;
      =     M   5265.7;
NETWORK
TITLE =

      AN    OV;
      =     L      0.0;
      A     L      0.0;
      AN    M   1900.0;
      =     M   5267.0;
      A     L      0.0;
      AN    M   1900.1;
      =     M   5267.1;
      A     L      0.0;
      A     M   1900.7;
      =     M   5267.2;
NETWORK
TITLE =
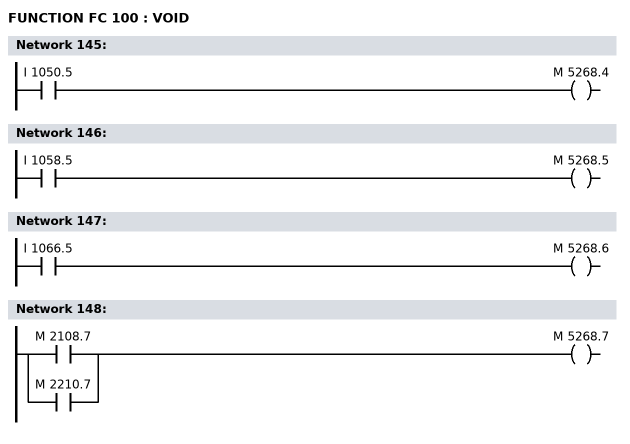

      A     I   1050.5;
      =     M   5268.4;
NETWORK
TITLE =

      A     I   1058.5;
      =     M   5268.5;
NETWORK
TITLE =

      A     I   1066.5;
      =     M   5268.6;
NETWORK
TITLE =

      O     M   2108.7;
      O     M   2210.7;
      =     M   5268.7;
NETWORK
TITLE =

      AN    OV;
      =     L      0.0;
      A     L      0.0;
      A(    ;
      O     M   2050.6;
      O     M   2050.7;
      )     ;
      =     M   5269.0;
      A     L      0.0;
      A(    ;
      O     M   2051.0;
      O     M   2051.1;
      )     ;
      =     M   5269.1;
      A     L      0.0;
      A(    ;
      O     M   2051.2;
      O     M   2051.3;
      )     ;
      =     M   5269.2;
NETWORK
TITLE =

      AN    OV;
      =     L      0.0;
      A     L      0.0;
      A     M   1506.5;
      =     M   5269.5;
      A     L      0.0;
      A     M   1506.6;
      =     M   5269.6;
      A     L      0.0;
      A     M   1506.7;
      =     M   5269.7;
END_FUNCTION

FUNCTION FC 101 : VOID
TITLE =
VERSION : 0.1

BEGIN
NETWORK
TITLE =
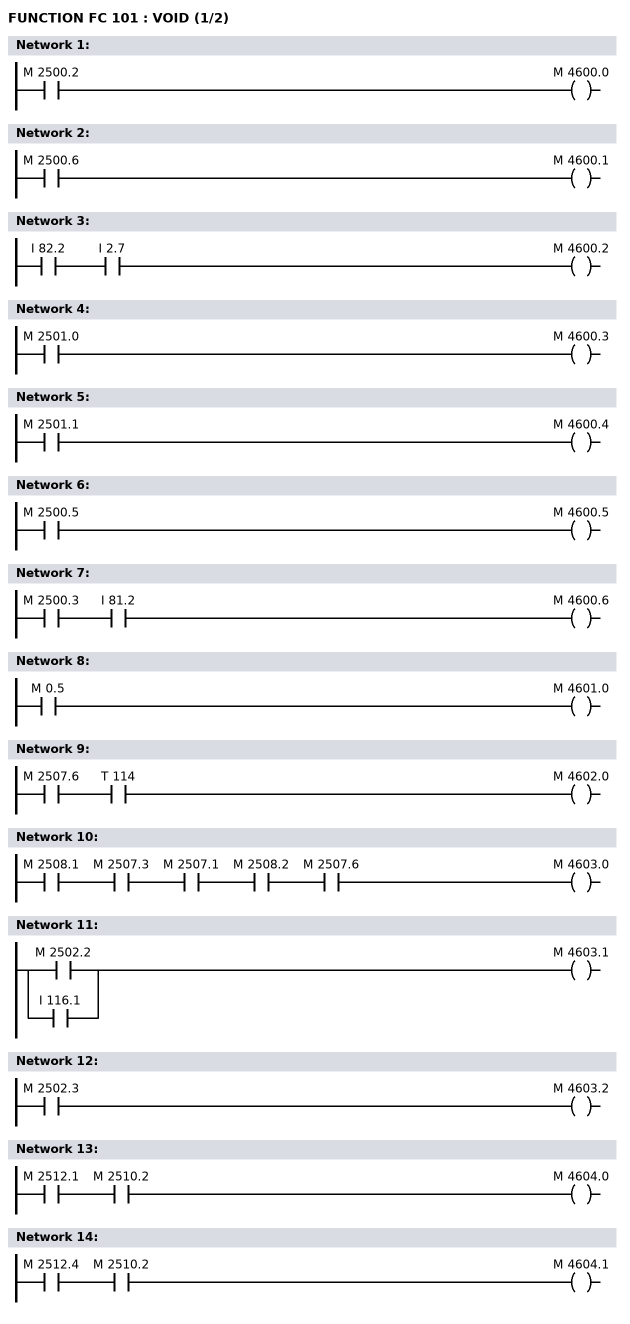

      A     M   2500.2;
      =     M   4600.0;
NETWORK
TITLE =

      A     M   2500.6;
      =     M   4600.1;
NETWORK
TITLE =

      A     I     82.2;
      A     I      2.7;
      =     M   4600.2;
NETWORK
TITLE =

      A     M   2501.0;
      =     M   4600.3;
NETWORK
TITLE =

      A     M   2501.1;
      =     M   4600.4;
NETWORK
TITLE =

      A     M   2500.5;
      =     M   4600.5;
NETWORK
TITLE =

      A     M   2500.3;
      A     I     81.2;
      =     M   4600.6;
NETWORK
TITLE =

      A     M      0.5;
      =     M   4601.0;
NETWORK
TITLE =

      A     M   2507.6;
      A     T    114;
      =     M   4602.0;
NETWORK
TITLE =

      A     M   2508.1;
      A     M   2507.3;
      A     M   2507.1;
      A     M   2508.2;
      A     M   2507.6;
      =     M   4603.0;
NETWORK
TITLE =

      O     M   2502.2;
      O     I    116.1;
      =     M   4603.1;
NETWORK
TITLE =

      A     M   2502.3;
      =     M   4603.2;
NETWORK
TITLE =

      A     M   2512.1;
      A     M   2510.2;
      =     M   4604.0;
NETWORK
TITLE =

      A     M   2512.4;
      A     M   2510.2;
      =     M   4604.1;
NETWORK
TITLE =
